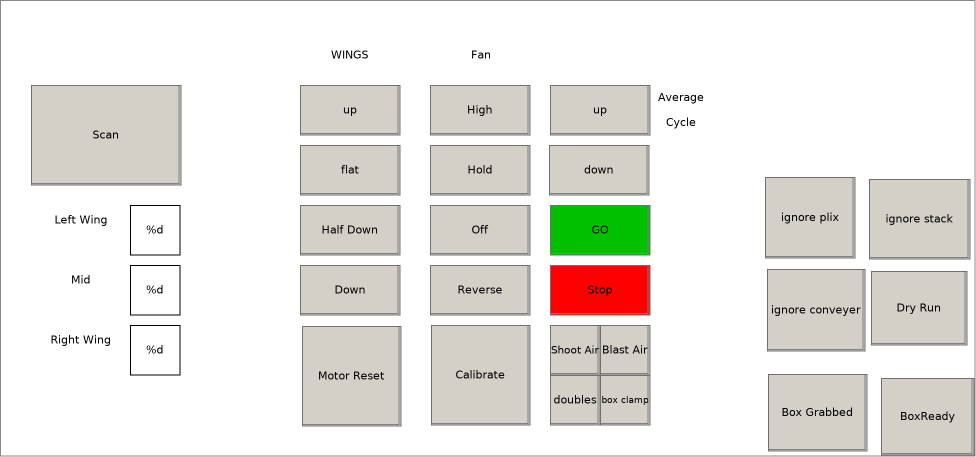
VISUALIZATION Visualization  // 976x457
    Button (31,85 150x100), "Scan"
        OnMouseDown: execute { GVL.ArduinoState := MAIN.PlixHandlerFB.Scanner; }
    Button (300,85 100x50), "up"
        OnMouseDown: execute { GVL.FanDyno := MAIN.PlixHandlerFB.WingUp; GVL.ArduinoState := MAIN.PlixHandlerFB.WingGo; }
    Button (300,145 100x50), "flat"
        OnMouseDown: execute { GVL.FanDyno := MAIN.PlixHandlerFB.WingFlat GVL.ArduinoState :=MAIN.PlixHandlerFB.WingGo }
    Button (300,265 100x50), "Down"
        OnMouseDown: execute { GVL.FanDyno :=MAIN.PlixHandlerFB.WingDown GVL.ArduinoState := MAIN.PlixHandlerFB.WingGo }
    Button (300,205 100x50), "Half Down"
        OnMouseDown: execute { GVL.FanDyno :=MAIN.PlixHandlerFB.WingHDown GVL.ArduinoState := MAIN.PlixHandlerFB.WingGo }
    Label (300,30 100x50), "WINGS"
    Button (430,85 100x50), "High"
        OnMouseDown: execute { GVL.FanDyno := MAIN.PlixHandlerFB.FanHigh; GVL.ArduinoState := MAIN.PlixHandlerFB.FanGo; }
    Button (430,205 100x50), "Off"
        OnMouseDown: execute { GVL.FanDyno :=MAIN.PlixHandlerFB.FanOff GVL.ArduinoState := MAIN.PlixHandlerFB.FanGo }
    Button (430,145 100x50), "Hold"
        OnMouseDown: execute { GVL.FanDyno :=MAIN.PlixHandlerFB.FanLow GVL.ArduinoState := MAIN.PlixHandlerFB.FanGo }
    Label (431,30 100x50), "Fan"
    Button (430,265 100x50), "Reverse"
        OnMouseDown: execute { GVL.FanDyno :=MAIN.PlixHandlerFB.FanReverse GVL.ArduinoState := MAIN.PlixHandlerFB.FanGo }
    Label (631,85 100x25), "Average"
    Label (631,110 100x25), "Cycle"
    Label (31,195 100x50), "Left Wing"
    Label (31,255 100x50), "Mid"
    Label (31,315 100x50), "Right Wing"
    Rectangle (130,205 50x50), "%d"
    Rectangle (130,265 50x50), "%d", text variable: GVL.Average
    Rectangle (130,325 50x50), "%d"
    Button (550,205 100x50), "GO"
        OnMouseUp: execute {
            MAIN.PlixHandlerFB.PlixHandlerState := 10;
            MAIN.GoTime := MAIN.TimeSeconds;
            MAIN.PlixHandlerFB.StackStepperHalt :=FALSE;
            MAIN.POUFB.BoxLoaderState :=100;
            MAIN.POUFB.FlapFolderState :=100;
            MAIN.POUFB.BoxRemoverState :=100;
            MAIN.POUFB.BoxRefillState :=100;
        }
    Button (550,265 100x50), "Stop"
        OnMouseDown: execute {
            MAIN.PlixHandlerFB.PlixHandlerState := 0;
            GVL.ArduinoState := 0;
            MAIN.PlixHandlerFB.StackStepperStop := TRUE;
            MAIN.PlixHandlerFB.StackStepperRun := FALSE;
            GVL.DoubleJets := FALSE;
            GVL.StackBlast := FALSE;
            GVL.PlixShooter := FALSE;
            MAIN.POUFB.BoxLoaderState :=0;
            MAIN.POUFB.FlapFolderState :=0;
            MAIN.POUFB.BoxRemoverState :=0;
            MAIN.TotalTime := MAIN.TimeSeconds;
        }
        OnMouseUp: execute { MAIN.PlixHandlerFB.StackStepperHalt :=FALSE; MAIN.PlixHandlerFB.Start :=TRUE; }
    Button (550,325 50x50), "Shoot Air"
        OnMouseDown: execute { GVL.PlixShooter := TRUE; }
        OnMouseUp: execute { GVL.PlixShooter := FALSE; }
    Button (600,325 50x50), "Blast Air"
        OnMouseDown: execute { GVL.StackBlast := TRUE; }
        OnMouseUp: execute { GVL.StackBlast := FALSE; }
    Button (550,85 100x50), "up"
    Button (549,145 100x50), "down"
    Button (550,375 50x50), "doubles"
        OnMouseDown: execute { GVL.DoubleJets := TRUE; }
        OnMouseUp: execute { GVL.DoubleJets := FALSE; }
    Button (600,375 50x50), "box clamp"
        OnMouseDown: execute { GVL.BottomClamp := TRUE; }
        OnMouseUp: execute { GVL.BottomClamp := FALSE; }
    Button (431,325 99x100), "Calibrate"
        OnMouseUp: execute { MAIN.PlixHandlerFB.Calibrate := TRUE; MAIN.PlixHandlerFB.PlixHandlerState := 10; }
    Button (302,326 99x100), "Motor Reset"
        OnMouseUp: execute { MAIN.PlixHandlerFB.StackStepperReset := FALSE; }
        OnMouseDown: execute { MAIN.PlixHandlerFB.StackStepperReset := TRUE; MAIN.PlixHandlerFB.StackStepperStop := FALSE; }
    Button (765,177 90x81), "ignore plix"
        OnMouseDown: execute { MAIN.POUFB.PlixRequest := FALSE; }
        OnMouseUp: execute {  }
    Button (869,179 101x80), "ignore stack"
        OnMouseDown: execute { MAIN.POUFB.BoxStackNeeded := FALSE; }
        OnMouseUp: execute {  }
    Button (767,269 98x82), "ignore conveyer"
        OnMouseDown: execute { MAIN.POUFB.BoxDropRequest := TRUE; MAIN.POUFB.BoxDropped := TRUE; }
    Button (871,271 96x74), "Dry Run"
        OnMouseDown: execute { MAIN.POUFB.DryRun := NOT MAIN.POUFB.DryRun }
    Button (768,374 99x77), "Box Grabbed"
        OnMouseDown: execute { MAIN.POUFB.BoxGrabbed := TRUE; MAIN.POUFB.BoxRemoved := TRUE; }
    Button (881,378 93x77), "BoxReady"
        OnMouseDown: execute { MAIN.POUFB.BoxReady := TRUE; }
END_VISUALIZATION

(* stored: Version 1.1.0.1, ProductVersion 3.1.4024.2
   Visu Visualization: Id {7ce1bdcb-bb5d-4f98-af3f-2564caddf423} *)
